(* IEC 61131-3 sources: Kur_TemplateProject_v1/TestPanelV1.fbsproj/MyController.device.xml.v3^/Plc Logic.plclogic.xml.v3^/Application.application.xml.v3^/Kur_Library/02_Blocks, 3 files *)

(* ---- AlarmSystem.fb.st ---- *)
FUNCTION_BLOCK AlarmSystem
VAR_INPUT
    Reset       : BOOL;
END_VAR
VAR_OUTPUT
    Active      : BOOL;                         // -> HMI lamp
    Count       : UINT;                         // -> HMI
    ActiveList  : ARRAY [1..20] OF UINT;        // -> HMI list
END_VAR
VAR
    Cond        : ARRAY [1..100] OF BOOL;
    Latch       : ARRAY [1..100] OF BOOL;
    ResetTrig   : R_TRIG;
    BuzzerTon   : TON;
    BuzzerLtc   : BOOL;
    i           : UINT;
    idx         : UINT;
END_VAR

// CALL LAST, AFTER ALL Chk() CALLS

ResetTrig(CLK := Reset);

Count := 0;
idx   := 0;

FOR i := 1 TO 100 DO

    // reset clears only alarms whose condition is gone
    IF ResetTrig.Q AND NOT Cond[i] THEN
        Latch[i] := FALSE;
    END_IF

    IF Latch[i] THEN
        Count := Count + 1;
        IF idx < 20 THEN
            idx := idx + 1;
            ActiveList[idx] := i;
        END_IF
    END_IF

END_FOR

FOR i := idx + 1 TO 20 DO
    ActiveList[i] := 0;
END_FOR

Active := (Count > 0);

IF ResetTrig.Q THEN
    BuzzerLtc := FALSE;
END_IF

BuzzerTon(IN := BuzzerLtc, PT := T#5S);

IF BuzzerTon.Q THEN
    BuzzerLtc := FALSE;
END_IF

(* ---- Button.fb.st ---- *)
FUNCTION_BLOCK Button

VAR_INPUT
    Signal : BOOL;        // Giriş sinyali
END_VAR

VAR_OUTPUT
    State      : BOOL;    // Anlık buton durumu
    Pressed    : BOOL;    // Basılma olayı (0 -> 1)
    Released  : BOOL;    // Bırakılma olayı (1 -> 0)
END_VAR

// Rising edge 0 -> 1
Pressed := Signal AND NOT State;

// Falling edge 1 -> 0
Released := NOT Signal AND State;

// Save Current state
State := Signal;

(* ---- EmergencyStop.fb.st ---- *)
FUNCTION_BLOCK EmergencyStop

VAR_INPUT
    Signal : BOOL;
END_VAR

VAR_OUTPUT
    OK : BOOL;		// when signal equal to TRUE.
    Active: BOOL;	// = True when signal is FALSE
END_VAR

OK := Signal;
Active := NOT Ok;
